// TwinCAT 3 PLC project TcSocketHelper_MultiServerString
// ProgramVersion: 3.1.0.5
// libraries:
//   Tc2_Standard, * (Beckhoff Automation GmbH)
//   Tc2_System, * (Beckhoff Automation GmbH)
//   Tc2_TcpIp, * (Beckhoff Automation GmbH)
//   Tc2_Utilities, * (Beckhoff Automation GmbH)
//   Tc3_Module, * (Beckhoff Automation GmbH)
// project tree:
//   Global Variables/ Global_Variables.TcGVL
//   POUs/ FB_Server.TcPOU, FB_ServerConnection.TcPOU, FB_ServerApplication.TcPOU, MAIN.TcPOU
//   POUs/Helper POUs/ FB_FrameFifo.TcPOU (not stored), FB_LogFifo.TcPOU (not stored)
//   / PlcTaskServer.TcTTO
// real-time tasks:
//   TASK PlcTaskServer: cycle T#10ms, priority 21, ADS port 351

CONFIGURATION TcSocketHelper_MultiServerString
    RESOURCE PLC ON TwinCAT3
        TASK PlcTaskServer(INTERVAL := T#10ms, PRIORITY := 21);
        PROGRAM MAIN WITH PlcTaskServer : MAIN;
    END_RESOURCE
END_CONFIGURATION

// ---- Global Variables/Global_Variables.TcGVL
VAR_GLOBAL CONSTANT
	PLCPRJ_BUFFER_SIZE						: UDINT := 1000;(* Max. internal fifo/receiver buffer size *)

(*	PLCPRJ_CLIENT_SEND_CYCLE_TIME			: TIME := T#1S; not used at server side *)
	PLCPRJ_RECEIVE_POLLING_TIME				: TIME := T#100MS;
	PLCPRJ_RECEIVE_TIMEOUT					: TIME := T#50S;

	(* Some project specific error codes *)
	PLCPRJ_ERROR_RECEIVE_TIMEOUT			: UDINT := 16#8101;(* Receive timeout *)
	PLCPRJ_ERROR_SENDFIFO_OVERFLOW			: UDINT := 16#8102;(* Send fifo overflow *)
	PLCPRJ_ERROR_RECFIFO_OVERFLOW			: UDINT := 16#8103;(* Receive fifo overflow *)
END_VAR

// ---- POUs/MAIN.TcPOU
PROGRAM MAIN
VAR
	sSrvNetID	: T_AmsNetID	:= '';(* TwinCAT TCP/IP server network address *)
	sLocalHost	: T_IPv4Addr	:= '127.0.0.1';(* Own (server) IP address! *)
	nLocalPort	: UDINT 		:= 200;(* Own (server) port number! *)
	bEnable1	: BOOL 			:= TRUE;(* TRUE => enable server (connection) instance, FALSE => disable *)
	bEnable2	: BOOL 			:= TRUE;
	bEnable3	: BOOL 			:= TRUE;
	bEnable4	: BOOL 			:= TRUE;
	bEnable5	: BOOL 			:= TRUE;
	bLog		: BOOL 			:= TRUE;(* TRUE => Enable error/message log, FALSE => Disable *)
	
	fbServer1	: FB_Server := ( sPrefix := 'SERVER1::' );(* Application (connection) instance *)
	fbServer2	: FB_Server := ( sPrefix := 'SERVER2::' );
	fbServer3	: FB_Server := ( sPrefix := 'SERVER3::' );
	fbServer4	: FB_Server := ( sPrefix := 'SERVER4::' );
	fbServer5	: FB_Server := ( sPrefix := 'SERVER5::' );
	hServer		: T_HSERVER;(* Server connection handle *)

	fbCloseAll	: FB_SocketCloseAll;
	bInitialize	: BOOL := TRUE;
END_VAR

(* On PLC reset or program download close all old (opened) connections *)
fbCloseAll( sSrvNetID := sSrvNetID, bExecute:= bInitialize );
IF fbCloseAll.bBusy OR fbCloseAll.bError THEN
	RETURN;
END_IF

IF bInitialize THEN
	bInitialize := FALSE;

	(* Initialize server handle *)
	F_CreateServerHnd( 	sSrvNetID 	:= sSrvNetID,
						sLocalHost 	:= sLocalHost,
						nLocalPort	:= nLocalPort,
						nMode 		:= SEL( bLog, 0, CONNECT_MODE_ENABLEDBG ),(* Enable/disable debug messages? *)
						bEnable 	:= FALSE,(* TRUE = leave listener socket open, FALSE = close listener socket after last connection ist closed too *)
						hServer 	:= hServer );
END_IF


(* Trigger the execution of every connection instance *)
fbServer1( hServer := hServer, sSrvNetID := sSrvNetID, bEnable := bEnable1, bLog := bLog );
fbServer2( hServer := hServer, sSrvNetID := sSrvNetID, bEnable := bEnable2, bLog := bLog );
fbServer3( hServer := hServer, sSrvNetID := sSrvNetID, bEnable := bEnable3, bLog := bLog );
fbServer4( hServer := hServer, sSrvNetID := sSrvNetID, bEnable := bEnable4, bLog := bLog );
fbServer5( hServer := hServer, sSrvNetID := sSrvNetID, bEnable := bEnable5, bLog := bLog );

END_PROGRAM

// ---- POUs/FB_Server.TcPOU
FUNCTION_BLOCK FB_Server
VAR_IN_OUT
	hServer			: T_HSERVER;(* Server connection handle *)
END_VAR
VAR_INPUT
	sSrvNetID		: T_AmsNetID	:= '';(* TwinCAT TCP/IP server network address *)
	bEnable			: BOOL 			:= FALSE;(* TRUE => enable server data exchange, FALSE => disable *)
	bLog			: BOOL 			:= FALSE;(* TRUE => Enable log message output, FALSE => Disable *)
	sPrefix			: STRING 		:= 'SERVER::';(* Log message description string (allows the identification of log message source) *)
END_VAR
VAR_OUTPUT
	eState			: E_SocketConnectionState := eSOCKET_DISCONNECTED;(* TCP/IP connection state *)
END_VAR
VAR
	fbApplication	: FB_ServerApplication;(* Server application control function block *)
	fbConnection	: FB_ServerConnection;(* Server data exchange control function block. Implements one server<->client connection *)
	fbTx 			: FB_FrameFifo;(* Tx fifo *)
	fbRx 			: FB_FrameFifo;(* Rx fifo *)
	fbLog			: FB_LogFifo;(* Log/debug/error fifo *)
END_VAR

(*-------------------------------- Trigger data exchange -----------------------------------------*)
fbConnection( hServer := hServer, sSrvNetID := sSrvNetID, fbRx := fbRx, fbTx := fbTx, fbLog := fbLog, 
			bEnable := bEnable, bLog := bLog, sPrefix := sPrefix, eState => eState );
IF fbConnection.eState = eSOCKET_CONNECTED THEN(* Connection established *)
	fbApplication( fbTx := fbTx, fbRx := fbRx, fbLog := fbLog );
END_IF

END_FUNCTION_BLOCK

// ---- POUs/FB_ServerApplication.TcPOU
(*----------------------- Simple TCP/IP application. Adapt this code to match your needs. ----*)
FUNCTION_BLOCK FB_ServerApplication
VAR_IN_OUT
	fbTx		: FB_FrameFifo;(* TX fifo *)
	fbRx		: FB_FrameFifo;(* RX fifo *)
	fbLog	 	: FB_LogFifo;(* Log/debug/error fifo *)
END_VAR
VAR
	sFromClient	: T_MaxString := '';
	sToClient	: T_MaxString := '';
	sLogMessage : T_MaxString := '';
	nCounter	: UDINT;
END_VAR

(*------------------------------- Get received message strings ------------------------------------------*)
REPEAT

	fbRx.RemoveHead( );(* Fetch received string from rx fifo *)
	IF fbRx.bOk THEN(* Success *)

		(*TODO: Implement receive data handler *)
		nCounter := nCounter + 1;
		sFromClient := fbRx.sGet;
		sToClient 	:= sFromClient;

		(* Send received string back to the client *)
		fbTx.AddTail( sPut := sToClient );(* Add string to the tx fifo *)
		IF NOT fbTx.bOk THEN(* Fifo overflow => log error *)
			fbLog.Error( sMessage := 'FB_FrameFifo(sender)', nErrID := PLCPRJ_ERROR_SENDFIFO_OVERFLOW );
		END_IF
	END_IF

UNTIL NOT fbRx.bOk
END_REPEAT



(*------------------------------- Get log/error messages from log fifo ----------------------------------------*)
REPEAT
	fbLog.Remove( );
	IF fbLog.bOk THEN

		(* TODO: Implement log message handler *)
		sLogMessage := fbLog.sGet;

	END_IF
UNTIL NOT fbLog.bOk
END_REPEAT

END_FUNCTION_BLOCK

// ---- POUs/FB_ServerConnection.TcPOU
(* This function block implements simple TCP/IP server protocol. *)
FUNCTION_BLOCK FB_ServerConnection
VAR_IN_OUT
	hServer		: T_HSERVER;(* Server connection handle *)
	fbTx		: FB_FrameFifo;(* TX fifo *)
	fbRx		: FB_FrameFifo;(* RX fifo *)
	fbLog	 	: FB_LogFifo;(* Log/debug/error fifo *)
END_VAR
VAR_INPUT
	sSrvNetID	: T_AmsNetID	:= '';(* TwinCAT TCP/IP server network address *)
	bEnable		: BOOL 			:= FALSE;(* TRUE => Enable/connect, FALSE => Disable/disconnect *)
	tReconnect 	: TIME 			:= T#1S;(* Try to reconnect after this time *)
	bLog		: BOOL 			:= FALSE;(* TRUE => Enable log message output, FALSE => Disable *)
	sPrefix		: STRING 		:= 'SERVER::';(* Log message description string (allows the identification of log message source) *)
END_VAR
VAR_OUTPUT
	eState		: E_SocketConnectionState := eSOCKET_DISCONNECTED;(* TCP/IP connection state *)
END_VAR
VAR
	fbConnect	: FB_ServerClientConnection;(* Create/release TCP/IP connection *)
	fbSend		: FB_SocketSend;(* Send TCP/IP data *)
	fbReceive	: FB_SocketReceive;(* Receive TCP/IP data *)
	nState 		: BYTE;(* Global state *)
	bSndBusy 	: BOOL;(* Tx state *)
	bRcvBusy 	: BOOL;(* Rx state *)
	bDisconnect	: BOOL;(* Disconnect flag, if set the socket will be closed *)

	fbPollTimer		: TON;(* Receive poll timer *)
	fbRequestTimer	: TON;(* Request timeout timer *)
	fbReconnectTimer : TON;(* Reconnect timer *)
	
	cbReceived	: UDINT;(* Count of received data bytes *)
	cbRx		: UDINT;(* Byte length of received string *)
	buffer		: ARRAY[0..PLCPRJ_BUFFER_SIZE] OF BYTE;(* Temp. RX buffer *)
	sTxFrame	: T_MaxString;
	sRxFrame	: T_MaxString;
	i			: UDINT;
	bAbort		: BOOL;
END_VAR

CASE nState OF
	0:(* Connect *)
		fbConnect( 	eMode := eACCEPT_ALL, tReconnect := tReconnect, bEnable := bEnable, 
					hServer := hServer, eState => eState );
		IF NOT fbConnect.bBusy THEN
			IF NOT fbConnect.bError THEN
				IF eState = eSOCKET_CONNECTED THEN(* We are connected *)

					fbTx.Clear( sPrefix := CONCAT( sPrefix, 'FB_FrameFifo(sender)::' ), bLog := bLog );(* Clear TX fifo (optional) *)
					fbRx.Clear( sPrefix := CONCAT( sPrefix, 'FB_FrameFifo(receiver)::' ), bLog := bLog );(* Clear RX fifo (optional) *)
					fbLog.Clear( sPrefix := sPrefix, bLog := bLog );(* Clear log fifo (optional) *)
					bSndBusy := FALSE;
					bRcvBusy := FALSE;
					bDisconnect := FALSE;
					cbReceived := 0;

					fbPollTimer( IN := FALSE, PT := T#0S );
					fbRequestTimer( IN := FALSE, PT := PLCPRJ_RECEIVE_TIMEOUT );
					fbReconnectTimer( IN := FALSE, PT := tReconnect );

					fbLog.Message( sMessage := 'Connection established!', hSocket := fbConnect.hSocket );
					nState := 1;
				END_IF
			ELSE(* Error => log error *)
				fbLog.Error( sMessage := 'FB_ServerClientConnection()', nErrID := fbConnect.nErrID );
			END_IF
		END_IF

	1:(* Data exchange state *)
		bDisconnect := NOT bEnable OR bDisconnect;(* User/internal disconnect requested? *)
		IF bDisconnect AND NOT bSndBusy AND NOT bRcvBusy THEN
			bDisconnect := FALSE;
			fbLog.Message( sMessage := 'Closing connection!', hSocket := fbConnect.hSocket );
			nState := 2;(* Disconnect *)
		ELSE

			(* ------------------------ Get rx data --------------------------------------- *)
			IF NOT bDisconnect AND NOT bRcvBusy THEN

				fbPollTimer( IN := TRUE );
				IF fbPollTimer.Q THEN
					IF fbRx.cbFree >= SIZEOF(sRxFrame) THEN(* Check free rx fifo space *)
						fbPollTimer( IN := FALSE, PT := PLCPRJ_RECEIVE_POLLING_TIME );
						fbReceive( bExecute := FALSE );
						fbReceive( sSrvNetId	:= sSrvNetID,
									hSocket		:= fbConnect.hSocket,
									cbLen		:= SIZEOF(buffer) - cbReceived,
									pDest		:= ADR(buffer) + cbReceived,
									bExecute	:= TRUE );
						bRcvBusy := TRUE;
					END_IF
				END_IF
				
			ELSE(* Wait until receive not busy *)
				
				fbReceive( bExecute := FALSE );
				IF NOT fbReceive.bBusy THEN
					bRcvBusy := FALSE;
					IF NOT fbReceive.bError THEN
						IF fbReceive.nRecBytes > 0 THEN(* Bytes received *)
							
							fbPollTimer( IN := FALSE, PT := T#0S );(* Bytes received => increase the read (polling) speed *)
							fbRequestTimer( IN := FALSE );(* Bytes received => disable timeout check *)
							cbReceived := cbReceived + fbReceive.nRecBytes;(* Calculate the number of received data bytes *)

							(* Parse received bytes and extract strings *)
							REPEAT
								bAbort := TRUE;(* Set flag *)
								IF cbReceived > 0 THEN

									(* Search for string null delimiter *)
									FOR i:= 0 TO cbReceived - 1 BY 1 DO
										IF buffer[i] = 0 THEN (* End of string position found *)

											cbRx := i + 1;(* Calculate the length of string (inclusive the end delimiter) *)
											MEMCPY( ADR(sRxFrame), ADR(buffer), MIN(cbRx, SIZEOF(sRxFrame) ) );(* Copy string bytes to fifo input variable *)

											fbRx.AddTail( sPut := sRxFrame );(* Add string to the rx fifo *)
											IF fbRx.bOk THEN

												MEMMOVE( ADR(buffer), ADR(buffer) + cbRx, cbReceived - cbRx );(* Move/shift remaining bytes in buffer *)
												cbReceived := cbReceived - cbRx;(* Recalculate the remaining data length *)

												IF fbRx.cbFree >= SIZEOF(sRxFrame) THEN(* Check free rx fifo space *)
													bAbort := FALSE;(* Reset flag, try to parse the next string  *)
												END_IF

											ELSE(* Fifo overflow => log error and disconnect *)
												fbLog.Error( sMessage := 'FB_FrameFifo(receiver)', nErrID := PLCPRJ_ERROR_RECFIFO_OVERFLOW );
												bDisconnect := TRUE;(* Set flag *)
												RETURN;
											END_IF

											EXIT;
										END_IF
									END_FOR

								END_IF (* IF cbReceived > 0 THEN *)

							UNTIL bAbort
							END_REPEAT

						ELSE(* No bytes received *)
							fbRequestTimer( IN := TRUE );(* No bytes received => enable timeout check *)
							IF fbRequestTimer.Q THEN (* Timeout error*)
								fbRequestTimer( IN := FALSE );
								fbLog.Error( sMessage := 'FB_SocketReceive()', nErrID := PLCPRJ_ERROR_RECEIVE_TIMEOUT );
								bDisconnect := TRUE;(* Set flag *)
							END_IF							
						END_IF(* IF fbReceive.nRecBytes > 0 THEN *)
					ELSE(* Receive error => log error and disconnect *)
						fbLog.Error( sMessage := 'FB_SocketReceive()', nErrID := fbReceive.nErrId );
						bDisconnect := TRUE;(* Set flag *)
					END_IF
				END_IF
			
			END_IF(* IF NOT bDisconnect AND NOT bRcvBusy THEN *)
			(* ---------------------------------------------------------------------------- *)


			(* --------------------------- Send tx data ----------------------------------- *)
			IF NOT bDisconnect AND NOT bSndBusy THEN
				fbTx.RemoveHead( sGet => sTxFrame );(* Remove oldest string entry s*)
				IF fbTx.bOk THEN(* Success *)
					fbSend( bExecute := FALSE );
					fbSend(	sSrvNetID 	:= sSrvNetID,
							hSocket		:= fbConnect.hSocket,
							cbLen		:= INT_TO_UDINT(LEN( sTxFrame )) + 1,(* Send string inclusive string (null) delimiter! *)
							pSrc		:= ADR( sTxFrame ),(* Address of the string variable *)
							bExecute	:= TRUE );
					bSndBusy := TRUE;
				END_IF
			ELSE(* Wait until send not busy *)
				fbSend( bExecute := FALSE );
				IF NOT fbSend.bBusy THEN
					bSndBusy := FALSE;
					IF fbSend.bError THEN(* Send error => log error and disconnect *)
						fbLog.Error( sMessage := 'FB_SocketSend()', nErrID := fbSend.nErrId );
						bDisconnect := TRUE;(* Set flag *)
					END_IF
				END_IF
			END_IF(* IF NOT bDisconnect AND NOT bSndBusy THEN *)
			(* ---------------------------------------------------------------------------- *)

			
		END_IF(* IF bDisconnect AND NOT bSndBusy AND NOT bRcvBusy THEN *)


	2:(* Disconnect *)
		fbConnect( hServer := hServer, bEnable:= FALSE, eState=>eState );
		IF eState = eSOCKET_DISCONNECTED THEN
			fbReconnectTimer( IN := TRUE );(* Please wait some seconds and then try to connect again *)
			IF fbReconnectTimer.Q THEN
				fbReconnectTimer( IN := FALSE );
				nState := 0;
			END_IF
		END_IF

END_CASE

END_FUNCTION_BLOCK
